Universal Robots PolyScope program: ros2_digital_pin_vacuum_control.urp

Program ros2_digital_pin_vacuum_control (installation=default directory=/programs/usbdisk createdIn=5.23.0 lastSavedIn=5.23.0 robotSerialNumber=20255701068)
Calibrated DH parameters: a=[0.000192, -0.240797, -0.145452, 0.000154, 0.000145, 0]; d=[0.162472, 156.092551, -478.083392, 322.124387, 0.099675, 0.09957]; alpha=[1.569919, -0.002247, 0.001132, 1.570007, -1.569568, 0]; deltaTheta=[0, -0.969163, -0.222039, 1.191203, 0, 0]
InitVariablesNode
Robot Program (runOnlyOnce=false)
  URCap External Control (External Control, FZI Research Center for Information Technology)
Thread Thread_2 (runOnlyOnce=false)
  Loop While (checkContinuously=false) expression=True
    If get_standard_digital_out(0) == True
      Script: rq_vacuum_grip( False, 60,40, 3000, True, "1" )
    ElseIf get_standard_digital_out( 0 ) == False
      Script: rq_vacuum_release( False, 5, True, "1" )
